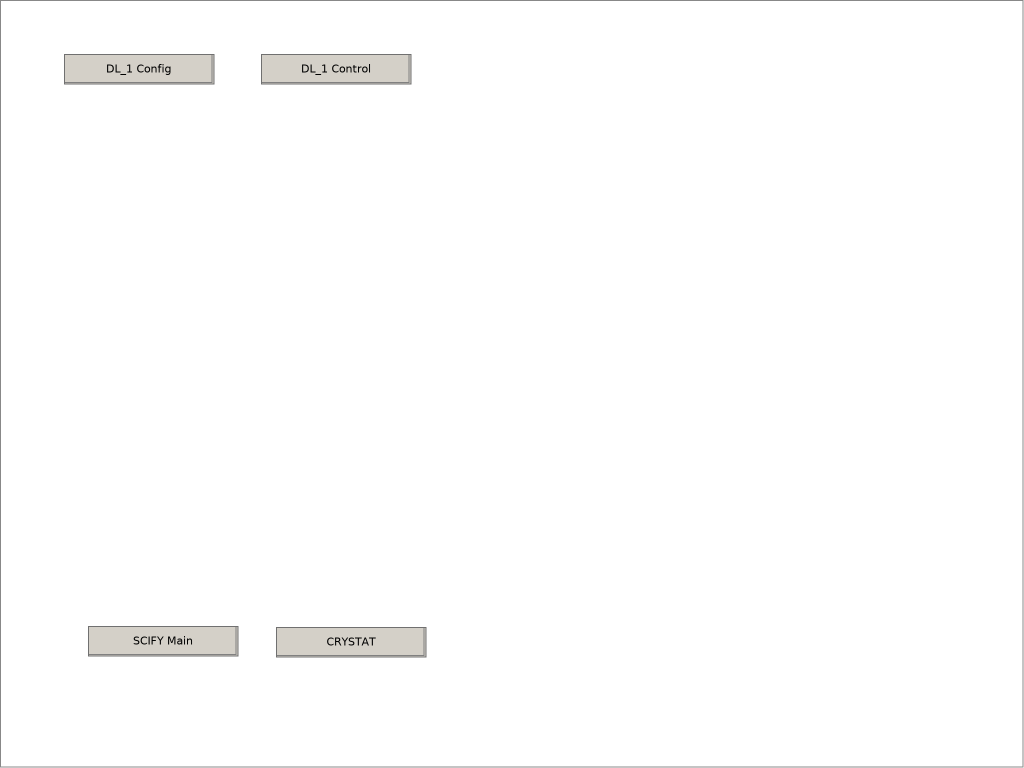
VISUALIZATION SCIFY_Delay_Lines  // 1024x768
    Button (88,626 150x30), "SCIFY Main"
        OnMouseDown: change screen: SCIFY_main
    Button (276,627 150x30), "CRYSTAT"
        OnMouseDown: change screen: SCIFY_Cryo
    Button (64,54 150x30), "DL_1 Config"
        OnMouseDown: change screen: DL_MOTOR_01_CONFIG
    Button (261,54 150x30), "DL_1 Control"
        OnMouseDown: change screen: DL_MOTOR_01_CTRL
END_VISUALIZATION

(* stored: Version 1.1.0.1, ProductVersion 3.1.4024.12
   Visu SCIFY_Delay_Lines: Id {a39198e8-f63a-4dde-88c2-cad7274a6fab} *)
